TYPE E_StateKompressor :
(
	eStateKompr_AUS,
	eStateKompr_START,
	eStateKompr_AKTIV,
	eStateKompr_STOP,
	eStateKompr_STOERUNG
);
END_TYPE

(* stored: Version 1.1.0.1, ProductVersion 3.1.4018.5
   DUT E_StateKompressor: Id {92d2eecc-4978-44ab-8abc-70d68f967281} *)
